INTERFACE ITF_Command

METHOD Execute : BOOL
VAR_INPUT
END_VAR
END_METHOD

END_INTERFACE

(* stored: Version 1.1.0.1, ProductVersion 3.1.4024.12
   Itf ITF_Command: Id {75e6c529-66b7-4e1f-992b-f40a85112a79}
   Method Execute: Id {cae199d4-de46-490e-9412-d6299fe62282} *)
